// TwinCAT 3 PLC project PLC1
// ProgramVersion: 3.1.4023.0
// libraries:
//   Tc2_Standard, * (Beckhoff Automation GmbH)
//   Tc2_System, * (Beckhoff Automation GmbH)
//   Tc3_Module, * (Beckhoff Automation GmbH)
// project tree:
//   / PlcTask.TcTTO
//   POUs/ MAIN.TcPOU
// real-time tasks:
//   TASK PlcTask: cycle T#10ms, priority 20, ADS port 350
// I/O:
//   DEVICE Device 1 (EtherCAT)
//     Term 1 (EK1100) [EK1100 EtherCAT Coupler (2A E-Bus)]
//       Term 2 (EL2008) [EL2008 8Ch. Dig. Output 24V, 0.5A]
//       Term 3 (EL2502) [EL2502 2Ch. PWM output, 24V]
// variable links:
//   PLC1/PLC1 Instance <-> Device 1 (EtherCAT)/Term 1 (EK1100)/Term 2 (EL2008)
//     PlcTask Outputs/MAIN.bOut[{0..7}] <-> Channel {1..8}/MAIN.bOut[{0..7}]  (8 links)

CONFIGURATION PLC1
    RESOURCE PLC ON TwinCAT3
        TASK PlcTask(INTERVAL := T#10ms, PRIORITY := 20);
        PROGRAM MAIN WITH PlcTask : MAIN;
    END_RESOURCE
END_CONFIGURATION

// ---- POUs/MAIN.TcPOU
PROGRAM MAIN
VAR
	bOut AT %Q*: ARRAY[0..7] OF BOOL;
	pwm AT %Q*: UINT;
	
END_VAR

pwm:=4000;

END_PROGRAM
